(* PLC project Montor Controller v1.0, D OpenPLC 1.0 *)
(* stored: creationDateTime 2018-09-26T00:48:44, modificationDateTime 2018-10-25T20:13:20 *)

PROGRAM Mixer_Control_Program
  VAR
    Motor_State AT %QX0.0 : BOOL;
  END_VAR
  VAR
    TMP : BOOL;
  END_VAR
  VAR
    Activation_Switch AT %QX1.3 : BOOL;
    Motor_Direction AT %QX0.1 : BOOL;
  END_VAR
  VAR
    TON1 : TON;
    TON2 : TON;
  END_VAR

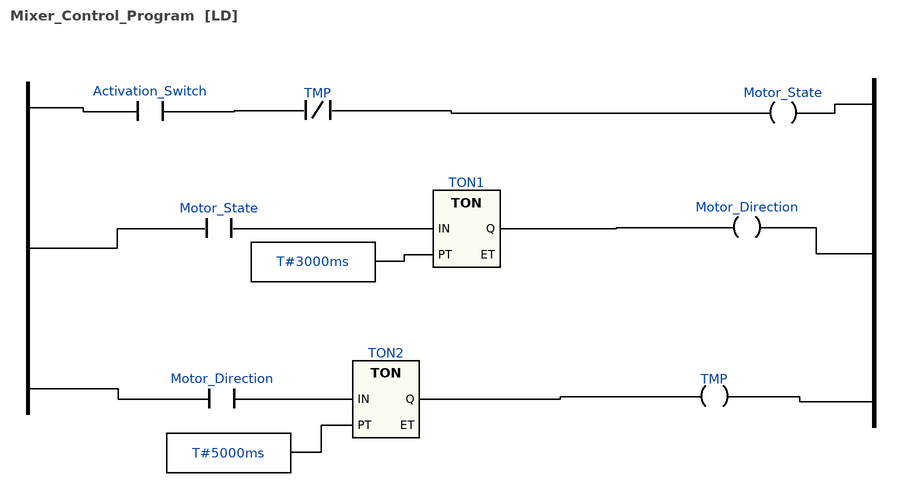
(* LD diagram, written out as Structured Text *)
Motor_State := Activation_Switch AND NOT TMP;
TON1(IN := Motor_State, PT := T#3000ms);
Motor_Direction := TON1.Q;
TON2(IN := Motor_Direction, PT := T#5000ms);
TMP := TON2.Q;
END_PROGRAM

PROGRAM Fan_Control_Program
  VAR
    Fan AT %QX0.2 : BOOL;
    Temperature AT %QW1 : INT := 0;
  END_VAR

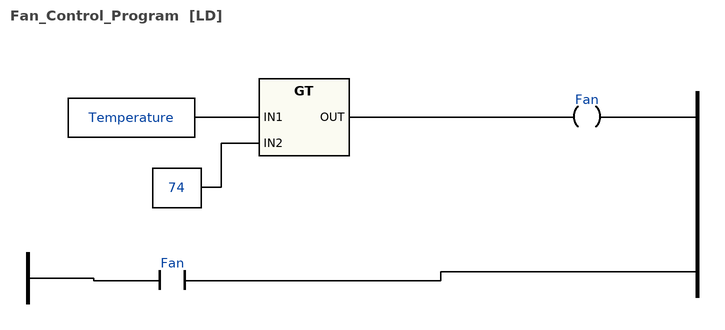
(* LD diagram, written out as Structured Text *)
Fan := Temperature > 74;
(* drawn but not wired to any output: Fan *)
END_PROGRAM

CONFIGURATION Config0
  RESOURCE Res0 ON PLC
    TASK ControlMotors(INTERVAL := T#50ms, PRIORITY := 0);
    TASK ControlFan(INTERVAL := T#50ms, PRIORITY := 0);
    PROGRAM instance0 WITH ControlMotors : Mixer_Control_Program;
    PROGRAM instance1 WITH ControlMotors : Fan_Control_Program;
  END_RESOURCE
END_CONFIGURATION
